(* IEC 61131-3 sources: nvidia-ai-factory-controls/tests/codesys/Safety, 1 file *)

(* ---- TEST_FB_EPO.fb ---- *)
(* =============================================================================
    TEST_FB_EPO — Unit Tests for Emergency Power Off Controller
    Test Library | NVIDIA AI Factory Controls
   ============================================================================= *)

FUNCTION_BLOCK TEST_FB_EPO EXTENDS FB_TestSuite
VAR
    _fbEPO               : FB_EPO_Controller;
    _i                   : INT;
END_VAR
